FUNCTION_BLOCK Motor_Direction
VAR_INPUT
	currentPositon: UINT;
	desiredPositon: UINT;
	writePostion: BOOL;
	positveMove: BOOL;
	negativeMove: BOOL;
	tolerance: UINT;
	
END_VAR
VAR_OUTPUT
	setPositveMove: BOOL;
	setNegativeMove: BOOL;
	setPositionCounter: UINT;
END_VAR
VAR
	referencePosition: UINT :=0;
END_VAR

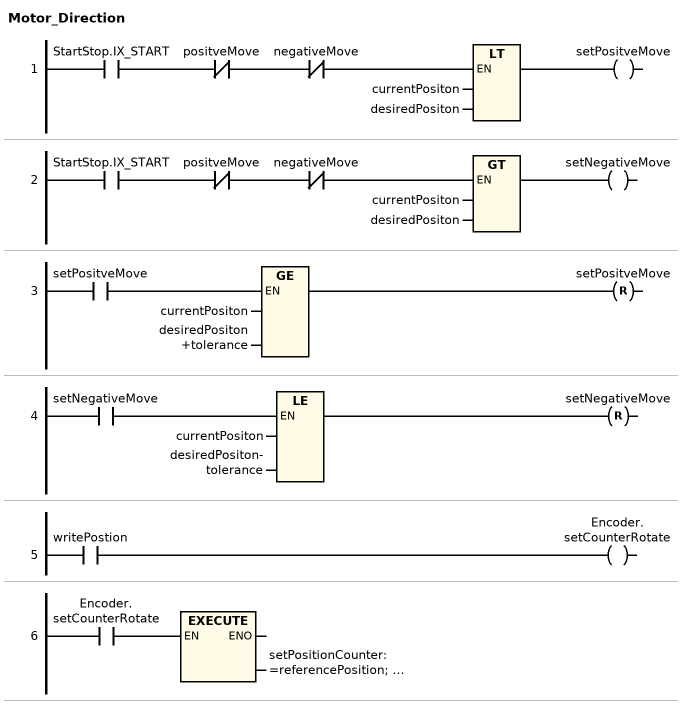
// NETWORK 1
setPositveMove := StartStop.IX_START AND NOT positveMove AND NOT negativeMove AND currentPositon < desiredPositon;

// NETWORK 2
setNegativeMove := StartStop.IX_START AND NOT positveMove AND NOT negativeMove AND currentPositon > desiredPositon;

// NETWORK 3
setPositveMove R= setPositveMove AND currentPositon >= (desiredPositon +tolerance);

// NETWORK 4
setNegativeMove R= setNegativeMove AND currentPositon <= (desiredPositon-tolerance);

// NETWORK 5
Encoder.setCounterRotate := writePostion;

// NETWORK 6
IF Encoder.setCounterRotate THEN setPositionCounter:=referencePosition; END_IF

END_FUNCTION_BLOCK

(* stored: Version 1.1.0.1, ProductVersion 3.1.4024.12
   POU Motor_Direction: Id {8fbc4570-101c-4e39-9754-c7aafbc7da5f}, SpecialFunc None *)
